FUNCTION_BLOCK S7_READ_CONTINUOUS_BYTE
  {SET_ATTRIBUTE(OpcUa, DEVICE.SENSOR)}
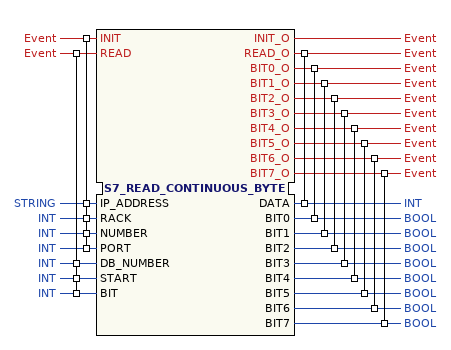
  EVENT_INPUT
    INIT WITH IP_ADDRESS, RACK, NUMBER, PORT;
    READ WITH DB_NUMBER, START, BIT;
  END_EVENT
  EVENT_OUTPUT
    INIT_O;
    READ_O WITH DATA;
    BIT0_O WITH BIT0;
    BIT1_O WITH BIT1;
    BIT2_O WITH BIT2;
    BIT3_O WITH BIT3;
    BIT4_O WITH BIT4;
    BIT5_O WITH BIT5;
    BIT6_O WITH BIT6;
    BIT7_O WITH BIT7;
  END_EVENT
  VAR_INPUT
    IP_ADDRESS : STRING; {SET_ATTRIBUTE(OpcUa, Constant.RUN)}
    RACK : INT; {SET_ATTRIBUTE(OpcUa, Constant.RUN)}
    NUMBER : INT; {SET_ATTRIBUTE(OpcUa, Constant.RUN)}
    PORT : INT; {SET_ATTRIBUTE(OpcUa, Constant.RUN)}
    DB_NUMBER : INT; {SET_ATTRIBUTE(OpcUa, Constant.RUN)}
    START : INT; {SET_ATTRIBUTE(OpcUa, Constant.RUN)}
    BIT : INT; {SET_ATTRIBUTE(OpcUa, Constant.RUN)}
  END_VAR
  VAR_OUTPUT
    DATA : INT; {SET_ATTRIBUTE(OpcUa, Variable.RUN)}
    BIT0 : BOOL; {SET_ATTRIBUTE(OpcUa, Variable.RUN)}
    BIT1 : BOOL; {SET_ATTRIBUTE(OpcUa, Variable.RUN)}
    BIT2 : BOOL; {SET_ATTRIBUTE(OpcUa, Variable.RUN)}
    BIT3 : BOOL; {SET_ATTRIBUTE(OpcUa, Variable.RUN)}
    BIT4 : BOOL; {SET_ATTRIBUTE(OpcUa, Variable.RUN)}
    BIT5 : BOOL; {SET_ATTRIBUTE(OpcUa, Variable.RUN)}
    BIT6 : BOOL; {SET_ATTRIBUTE(OpcUa, Variable.RUN)}
    BIT7 : BOOL; {SET_ATTRIBUTE(OpcUa, Variable.RUN)}
  END_VAR
END_FUNCTION_BLOCK
